// TIA Portal V20 export
// export: Created 2025-12-01T14:56:17.5233973Z, ExportSetting None, DisplayName Totally Integrated Automation Portal, DisplayVersion V20 Update 3, DisplayName TIA Portal Openness, DisplayVersion V20 Update 3, DisplayName TIA Portal Version Control Interface, DisplayVersion V20 Update 3, DisplayName STEP 7 Professional, DisplayVersion V20 Update 3, DisplayName STEP 7 Safety, DisplayVersion V20 Update 2, DisplayName WinCC Basic/Comfort/Advanced, DisplayVersion V20 Update 3, DisplayName WinCC Professional, DisplayVersion V20 Update 3, DisplayName WinCC Unified, DisplayVersion V20 Update 3
TYPE "Interlock_QubiqaUlma"
   STRUCT
      TL_Online { ExternalVisible := 'False'} : Bool;
      TL_Alive { ExternalVisible := 'False'} : Bool;
      TL1_Run { ExternalVisible := 'False'} : Bool;
      TL2_Run { ExternalVisible := 'False'} : Bool;
      TL1_StartButton { ExternalVisible := 'False'} : Bool;
      TL1_ResetButton { ExternalVisible := 'False'} : Bool;
      TL2_StartButton { ExternalVisible := 'False'} : Bool;
      TL2_ResetButton { ExternalVisible := 'False'} : Bool;
      Reserve_1_0 { ExternalVisible := 'False'} : Bool;
      Reserve_1_1 { ExternalVisible := 'False'} : Bool;
      Reserve_1_2 { ExternalVisible := 'False'} : Bool;
      Reserve_1_3 { ExternalVisible := 'False'} : Bool;
      Reserve_1_4 { ExternalVisible := 'False'} : Bool;
      Reserve_1_5 { ExternalVisible := 'False'} : Bool;
      Reserve_1_6 { ExternalVisible := 'False'} : Bool;
      Reserve_1_7 { ExternalVisible := 'False'} : Bool;
      LineRunning_L1 { ExternalVisible := 'False'} : Bool;
      TrayInTransfer_L1 { ExternalVisible := 'False'} : Bool;
      SorterInductionSpeed_L1 { ExternalVisible := 'False'} : Bool;
      SizeControl_L1 { ExternalVisible := 'False'} : Bool;
      Reserve_2_4 { ExternalVisible := 'False'} : Bool;
      Reserve_2_5 { ExternalVisible := 'False'} : Bool;
      Reserve_2_6 { ExternalVisible := 'False'} : Bool;
      OrderFinished_L1 { ExternalVisible := 'False'} : Bool;
      PermissionToSend_L1 { ExternalVisible := 'False'} : Bool;
      TranserFinished_L1 { ExternalVisible := 'False'} : Bool;
      OrderFinished_Ok_L1 { ExternalVisible := 'False'} : Bool;
      reserva_3_3 { ExternalVisible := 'False'} : Bool;
      reserva_3_4 { ExternalVisible := 'False'} : Bool;
      reserva_3_5 { ExternalVisible := 'False'} : Bool;
      reserva_3_6 { ExternalVisible := 'False'} : Bool;
      reserva_3_7 { ExternalVisible := 'False'} : Bool;
      StartStack_Small_L1 { ExternalVisible := 'False'} : Bool;
      StackReceived_Small_L1 { ExternalVisible := 'False'} : Bool;
      reserva_4_2 { ExternalVisible := 'False'} : Bool;
      reserva_4_3 { ExternalVisible := 'False'} : Bool;
      reserva_4_4 { ExternalVisible := 'False'} : Bool;
      reserva_4_5 { ExternalVisible := 'False'} : Bool;
      reserva_4_6 { ExternalVisible := 'False'} : Bool;
      reserva_4_7 { ExternalVisible := 'False'} : Bool;
      NoStackInBuffer_Small_L1 { ExternalVisible := 'False'} : Byte;
      StartStack_Large_L1 { ExternalVisible := 'False'} : Bool;
      StackReceived_Large_L1 { ExternalVisible := 'False'} : Bool;
      reserva_6_2 { ExternalVisible := 'False'} : Bool;
      reserva_6_3 { ExternalVisible := 'False'} : Bool;
      reserva_6_4 { ExternalVisible := 'False'} : Bool;
      reserva_6_5 { ExternalVisible := 'False'} : Bool;
      reserva_6_6 { ExternalVisible := 'False'} : Bool;
      reserva_6_7 { ExternalVisible := 'False'} : Bool;
      NoStackInBuffer_Large_L1 { ExternalVisible := 'False'} : Byte;
      reserva_8_0 { ExternalVisible := 'False'} : Bool;
      reserva_8_1 { ExternalVisible := 'False'} : Bool;
      reserva_8_2 { ExternalVisible := 'False'} : Bool;
      reserva_8_3 { ExternalVisible := 'False'} : Bool;
      reserva_8_4 { ExternalVisible := 'False'} : Bool;
      reserva_8_5 { ExternalVisible := 'False'} : Bool;
      reserva_8_6 { ExternalVisible := 'False'} : Bool;
      reserva_8_7 { ExternalVisible := 'False'} : Bool;
      reserva_9_0 { ExternalVisible := 'False'} : Bool;
      reserva_9_1 { ExternalVisible := 'False'} : Bool;
      reserva_9_2 { ExternalVisible := 'False'} : Bool;
      reserva_9_3 { ExternalVisible := 'False'} : Bool;
      reserva_9_4 { ExternalVisible := 'False'} : Bool;
      reserva_9_5 { ExternalVisible := 'False'} : Bool;
      reserva_9_6 { ExternalVisible := 'False'} : Bool;
      reserva_9_7 { ExternalVisible := 'False'} : Bool;
      LineRunning_L2 { ExternalVisible := 'False'} : Bool;
      TrayInTransfer_L2 { ExternalVisible := 'False'} : Bool;
      SorterInductionSpeed_L2 { ExternalVisible := 'False'} : Bool;
      SizeControl_L2 { ExternalVisible := 'False'} : Bool;
      reserva_10_4 { ExternalVisible := 'False'} : Bool;
      reserva_10_5 { ExternalVisible := 'False'} : Bool;
      reserva_10_6 { ExternalVisible := 'False'} : Bool;
      OrderFinished_L2 { ExternalVisible := 'False'} : Bool;
      PermissionToSend_L2 { ExternalVisible := 'False'} : Bool;
      TranserFinished_L2 { ExternalVisible := 'False'} : Bool;
      OrderFinished_Ok_L2 { ExternalVisible := 'False'} : Bool;
      reserva_11_3 { ExternalVisible := 'False'} : Bool;
      reserva_11_4 { ExternalVisible := 'False'} : Bool;
      reserva_11_5 { ExternalVisible := 'False'} : Bool;
      reserva_11_6 { ExternalVisible := 'False'} : Bool;
      reserva_11_7 { ExternalVisible := 'False'} : Bool;
      StartStack_Small_L2 { ExternalVisible := 'False'} : Bool;
      StackReceived_Small_L2 { ExternalVisible := 'False'} : Bool;
      reserva_12_2 { ExternalVisible := 'False'} : Bool;
      reserva_12_3 { ExternalVisible := 'False'} : Bool;
      reserva_12_4 { ExternalVisible := 'False'} : Bool;
      reserva_12_5 { ExternalVisible := 'False'} : Bool;
      reserva_12_6 { ExternalVisible := 'False'} : Bool;
      reserva_12_7 { ExternalVisible := 'False'} : Bool;
      NoStackInBuffer_Small_L2 { ExternalVisible := 'False'} : Byte;
      StartStack_Large_L2 { ExternalVisible := 'False'} : Bool;
      StackReceived_Large_L2 { ExternalVisible := 'False'} : Bool;
      reserva_14_2 { ExternalVisible := 'False'} : Bool;
      reserva_14_3 { ExternalVisible := 'False'} : Bool;
      reserva_14_4 { ExternalVisible := 'False'} : Bool;
      reserva_14_5 { ExternalVisible := 'False'} : Bool;
      reserva_14_6 { ExternalVisible := 'False'} : Bool;
      reserva_14_7 { ExternalVisible := 'False'} : Bool;
      NoStackInBuffer_Large_L2 { ExternalVisible := 'False'} : Byte;
      reserva_16_0 { ExternalVisible := 'False'} : Bool;
      reserva_16_1 { ExternalVisible := 'False'} : Bool;
      reserva_16_2 { ExternalVisible := 'False'} : Bool;
      reserva_16_3 { ExternalVisible := 'False'} : Bool;
      reserva_16_4 { ExternalVisible := 'False'} : Bool;
      reserva_16_5 { ExternalVisible := 'False'} : Bool;
      reserva_16_6 { ExternalVisible := 'False'} : Bool;
      reserva_16_7 { ExternalVisible := 'False'} : Bool;
      reserva_17_0 { ExternalVisible := 'False'} : Bool;
      reserva_17_1 { ExternalVisible := 'False'} : Bool;
      reserva_17_2 { ExternalVisible := 'False'} : Bool;
      reserva_17_3 { ExternalVisible := 'False'} : Bool;
      reserva_17_4 { ExternalVisible := 'False'} : Bool;
      reserva_17_5 { ExternalVisible := 'False'} : Bool;
      reserva_17_6 { ExternalVisible := 'False'} : Bool;
      reserva_17_7 { ExternalVisible := 'False'} : Bool;
      reserva_18_0 { ExternalVisible := 'False'} : Bool;
      reserva_18_1 { ExternalVisible := 'False'} : Bool;
      reserva_18_2 { ExternalVisible := 'False'} : Bool;
      reserva_18_3 { ExternalVisible := 'False'} : Bool;
      reserva_18_4 { ExternalVisible := 'False'} : Bool;
      reserva_18_5 { ExternalVisible := 'False'} : Bool;
      reserva_18_6 { ExternalVisible := 'False'} : Bool;
      reserva_18_7 { ExternalVisible := 'False'} : Bool;
      reserva_19_0 { ExternalVisible := 'False'} : Bool;
      reserva_19_1 { ExternalVisible := 'False'} : Bool;
      reserva_19_2 { ExternalVisible := 'False'} : Bool;
      reserva_19_3 { ExternalVisible := 'False'} : Bool;
      reserva_19_4 { ExternalVisible := 'False'} : Bool;
      reserva_19_5 { ExternalVisible := 'False'} : Bool;
      reserva_19_6 { ExternalVisible := 'False'} : Bool;
      reserva_19_7 { ExternalVisible := 'False'} : Bool;
      reserva_20_0 { ExternalVisible := 'False'} : Bool;
      reserva_20_1 { ExternalVisible := 'False'} : Bool;
      reserva_20_2 { ExternalVisible := 'False'} : Bool;
      reserva_20_3 { ExternalVisible := 'False'} : Bool;
      reserva_20_4 { ExternalVisible := 'False'} : Bool;
      reserva_20_5 { ExternalVisible := 'False'} : Bool;
      reserva_20_6 { ExternalVisible := 'False'} : Bool;
      reserva_20_7 { ExternalVisible := 'False'} : Bool;
      reserva_21_0 { ExternalVisible := 'False'} : Bool;
      reserva_21_1 { ExternalVisible := 'False'} : Bool;
      reserva_21_2 { ExternalVisible := 'False'} : Bool;
      reserva_21_3 { ExternalVisible := 'False'} : Bool;
      reserva_21_4 { ExternalVisible := 'False'} : Bool;
      reserva_21_5 { ExternalVisible := 'False'} : Bool;
      reserva_21_6 { ExternalVisible := 'False'} : Bool;
      reserva_21_7 { ExternalVisible := 'False'} : Bool;
      reserva_22_0 { ExternalVisible := 'False'} : Bool;
      reserva_22_1 { ExternalVisible := 'False'} : Bool;
      reserva_22_2 { ExternalVisible := 'False'} : Bool;
      reserva_22_3 { ExternalVisible := 'False'} : Bool;
      reserva_22_4 { ExternalVisible := 'False'} : Bool;
      reserva_22_5 { ExternalVisible := 'False'} : Bool;
      reserva_22_6 { ExternalVisible := 'False'} : Bool;
      reserva_22_7 { ExternalVisible := 'False'} : Bool;
      reserva_23_0 { ExternalVisible := 'False'} : Bool;
      reserva_23_1 { ExternalVisible := 'False'} : Bool;
      reserva_23_2 { ExternalVisible := 'False'} : Bool;
      reserva_23_3 { ExternalVisible := 'False'} : Bool;
      reserva_23_4 { ExternalVisible := 'False'} : Bool;
      reserva_23_5 { ExternalVisible := 'False'} : Bool;
      reserva_23_6 { ExternalVisible := 'False'} : Bool;
      reserva_23_7 { ExternalVisible := 'False'} : Bool;
      reserva_24_0 { ExternalVisible := 'False'} : Bool;
      reserva_24_1 { ExternalVisible := 'False'} : Bool;
      reserva_24_2 { ExternalVisible := 'False'} : Bool;
      reserva_24_3 { ExternalVisible := 'False'} : Bool;
      reserva_24_4 { ExternalVisible := 'False'} : Bool;
      reserva_24_5 { ExternalVisible := 'False'} : Bool;
      reserva_24_6 { ExternalVisible := 'False'} : Bool;
      reserva_24_7 { ExternalVisible := 'False'} : Bool;
      reserva_25_0 { ExternalVisible := 'False'} : Bool;
      reserva_25_1 { ExternalVisible := 'False'} : Bool;
      reserva_25_2 { ExternalVisible := 'False'} : Bool;
      reserva_25_3 { ExternalVisible := 'False'} : Bool;
      reserva_25_4 { ExternalVisible := 'False'} : Bool;
      reserva_25_5 { ExternalVisible := 'False'} : Bool;
      reserva_25_6 { ExternalVisible := 'False'} : Bool;
      reserva_25_7 { ExternalVisible := 'False'} : Bool;
      reserva_26_0 { ExternalVisible := 'False'} : Bool;
      reserva_26_1 { ExternalVisible := 'False'} : Bool;
      reserva_26_2 { ExternalVisible := 'False'} : Bool;
      reserva_26_3 { ExternalVisible := 'False'} : Bool;
      reserva_26_4 { ExternalVisible := 'False'} : Bool;
      reserva_26_5 { ExternalVisible := 'False'} : Bool;
      reserva_26_6 { ExternalVisible := 'False'} : Bool;
      reserva_26_7 { ExternalVisible := 'False'} : Bool;
      reserva_27_0 { ExternalVisible := 'False'} : Bool;
      reserva_27_1 { ExternalVisible := 'False'} : Bool;
      reserva_27_2 { ExternalVisible := 'False'} : Bool;
      reserva_27_3 { ExternalVisible := 'False'} : Bool;
      reserva_27_4 { ExternalVisible := 'False'} : Bool;
      reserva_27_5 { ExternalVisible := 'False'} : Bool;
      reserva_27_6 { ExternalVisible := 'False'} : Bool;
      reserva_27_7 { ExternalVisible := 'False'} : Bool;
      reserva_28_0 { ExternalVisible := 'False'} : Bool;
      reserva_28_1 { ExternalVisible := 'False'} : Bool;
      reserva_28_2 { ExternalVisible := 'False'} : Bool;
      reserva_28_3 { ExternalVisible := 'False'} : Bool;
      reserva_28_4 { ExternalVisible := 'False'} : Bool;
      reserva_28_5 { ExternalVisible := 'False'} : Bool;
      reserva_28_6 { ExternalVisible := 'False'} : Bool;
      reserva_28_7 { ExternalVisible := 'False'} : Bool;
      reserva_29_0 { ExternalVisible := 'False'} : Bool;
      reserva_29_1 { ExternalVisible := 'False'} : Bool;
      reserva_29_2 { ExternalVisible := 'False'} : Bool;
      reserva_29_3 { ExternalVisible := 'False'} : Bool;
      reserva_29_4 { ExternalVisible := 'False'} : Bool;
      reserva_29_5 { ExternalVisible := 'False'} : Bool;
      reserva_29_6 { ExternalVisible := 'False'} : Bool;
      reserva_29_7 { ExternalVisible := 'False'} : Bool;
      Reserve_30_0 { ExternalVisible := 'False'} : Bool;
      Reserve_30_1 { ExternalVisible := 'False'} : Bool;
      Reserve_30_2 { ExternalVisible := 'False'} : Bool;
      Reserve_30_3 { ExternalVisible := 'False'} : Bool;
      Reserve_30_4 { ExternalVisible := 'False'} : Bool;
      Reserve_30_5 { ExternalVisible := 'False'} : Bool;
      Reserve_30_6 { ExternalVisible := 'False'} : Bool;
      Reserve_30_7 { ExternalVisible := 'False'} : Bool;
      Reserve_31_0 { ExternalVisible := 'False'} : Bool;
      Reserve_31_1 { ExternalVisible := 'False'} : Bool;
      Reserve_31_2 { ExternalVisible := 'False'} : Bool;
      Reserve_31_3 { ExternalVisible := 'False'} : Bool;
      Reserve_31_4 { ExternalVisible := 'False'} : Bool;
      Reserve_31_5 { ExternalVisible := 'False'} : Bool;
      Reserve_31_6 { ExternalVisible := 'False'} : Bool;
      Reserve_31_7 { ExternalVisible := 'False'} : Bool;
      Reserve_32_0 { ExternalVisible := 'False'} : Bool;
      Reserve_32_1 { ExternalVisible := 'False'} : Bool;
      Reserve_32_2 { ExternalVisible := 'False'} : Bool;
      Reserve_32_3 { ExternalVisible := 'False'} : Bool;
      Reserve_32_4 { ExternalVisible := 'False'} : Bool;
      Reserve_32_5 { ExternalVisible := 'False'} : Bool;
      Reserve_32_6 { ExternalVisible := 'False'} : Bool;
      Reserve_32_7 { ExternalVisible := 'False'} : Bool;
      reserva_33_0 { ExternalVisible := 'False'} : Bool;
      reserva_33_1 { ExternalVisible := 'False'} : Bool;
      reserva_33_2 { ExternalVisible := 'False'} : Bool;
      reserva_33_3 { ExternalVisible := 'False'} : Bool;
      reserva_33_4 { ExternalVisible := 'False'} : Bool;
      reserva_33_5 { ExternalVisible := 'False'} : Bool;
      reserva_33_6 { ExternalVisible := 'False'} : Bool;
      reserva_33_7 { ExternalVisible := 'False'} : Bool;
      reserva_34_0 { ExternalVisible := 'False'} : Bool;
      reserva_34_1 { ExternalVisible := 'False'} : Bool;
      reserva_34_2 { ExternalVisible := 'False'} : Bool;
      reserva_34_3 { ExternalVisible := 'False'} : Bool;
      reserva_34_4 { ExternalVisible := 'False'} : Bool;
      reserva_34_5 { ExternalVisible := 'False'} : Bool;
      reserva_34_6 { ExternalVisible := 'False'} : Bool;
      reserva_34_7 { ExternalVisible := 'False'} : Bool;
      reserva_35_0 { ExternalVisible := 'False'} : Bool;
      reserva_35_1 { ExternalVisible := 'False'} : Bool;
      reserva_35_2 { ExternalVisible := 'False'} : Bool;
      reserva_35_3 { ExternalVisible := 'False'} : Bool;
      reserva_35_4 { ExternalVisible := 'False'} : Bool;
      reserva_35_5 { ExternalVisible := 'False'} : Bool;
      reserva_35_6 { ExternalVisible := 'False'} : Bool;
      reserva_35_7 { ExternalVisible := 'False'} : Bool;
      reserva_36_0 { ExternalVisible := 'False'} : Bool;
      reserva_36_1 { ExternalVisible := 'False'} : Bool;
      reserva_36_2 { ExternalVisible := 'False'} : Bool;
      reserva_36_3 { ExternalVisible := 'False'} : Bool;
      reserva_36_4 { ExternalVisible := 'False'} : Bool;
      reserva_36_5 { ExternalVisible := 'False'} : Bool;
      reserva_36_6 { ExternalVisible := 'False'} : Bool;
      reserva_36_7 { ExternalVisible := 'False'} : Bool;
      reserva_37_0 { ExternalVisible := 'False'} : Bool;
      reserva_37_1 { ExternalVisible := 'False'} : Bool;
      reserva_37_2 { ExternalVisible := 'False'} : Bool;
      reserva_37_3 { ExternalVisible := 'False'} : Bool;
      reserva_37_4 { ExternalVisible := 'False'} : Bool;
      reserva_37_5 { ExternalVisible := 'False'} : Bool;
      reserva_37_6 { ExternalVisible := 'False'} : Bool;
      reserva_37_7 { ExternalVisible := 'False'} : Bool;
      reserva_38_0 { ExternalVisible := 'False'} : Bool;
      reserva_38_1 { ExternalVisible := 'False'} : Bool;
      reserva_38_2 { ExternalVisible := 'False'} : Bool;
      reserva_38_3 { ExternalVisible := 'False'} : Bool;
      reserva_38_4 { ExternalVisible := 'False'} : Bool;
      reserva_38_5 { ExternalVisible := 'False'} : Bool;
      reserva_38_6 { ExternalVisible := 'False'} : Bool;
      reserva_38_7 { ExternalVisible := 'False'} : Bool;
      reserva_39_0 { ExternalVisible := 'False'} : Bool;
      reserva_39_1 { ExternalVisible := 'False'} : Bool;
      reserva_39_2 { ExternalVisible := 'False'} : Bool;
      reserva_39_3 { ExternalVisible := 'False'} : Bool;
      reserva_39_4 { ExternalVisible := 'False'} : Bool;
      reserva_39_5 { ExternalVisible := 'False'} : Bool;
      reserva_39_6 { ExternalVisible := 'False'} : Bool;
      reserva_39_7 { ExternalVisible := 'False'} : Bool;
      reserva_40_0 { ExternalVisible := 'False'} : Bool;
      reserva_40_1 { ExternalVisible := 'False'} : Bool;
      reserva_40_2 { ExternalVisible := 'False'} : Bool;
      reserva_40_3 { ExternalVisible := 'False'} : Bool;
      reserva_40_4 { ExternalVisible := 'False'} : Bool;
      reserva_40_5 { ExternalVisible := 'False'} : Bool;
      reserva_40_6 { ExternalVisible := 'False'} : Bool;
      reserva_40_7 { ExternalVisible := 'False'} : Bool;
      reserva_41_0 { ExternalVisible := 'False'} : Bool;
      reserva_41_1 { ExternalVisible := 'False'} : Bool;
      reserva_41_2 { ExternalVisible := 'False'} : Bool;
      reserva_41_3 { ExternalVisible := 'False'} : Bool;
      reserva_41_4 { ExternalVisible := 'False'} : Bool;
      reserva_41_5 { ExternalVisible := 'False'} : Bool;
      reserva_41_6 { ExternalVisible := 'False'} : Bool;
      reserva_41_7 { ExternalVisible := 'False'} : Bool;
      reserva_42_0 { ExternalVisible := 'False'} : Bool;
      reserva_42_1 { ExternalVisible := 'False'} : Bool;
      reserva_42_2 { ExternalVisible := 'False'} : Bool;
      reserva_42_3 { ExternalVisible := 'False'} : Bool;
      reserva_42_4 { ExternalVisible := 'False'} : Bool;
      reserva_42_5 { ExternalVisible := 'False'} : Bool;
      reserva_42_6 { ExternalVisible := 'False'} : Bool;
      reserva_42_7 { ExternalVisible := 'False'} : Bool;
      reserva_43_0 { ExternalVisible := 'False'} : Bool;
      reserva_43_1 { ExternalVisible := 'False'} : Bool;
      reserva_43_2 { ExternalVisible := 'False'} : Bool;
      reserva_43_3 { ExternalVisible := 'False'} : Bool;
      reserva_43_4 { ExternalVisible := 'False'} : Bool;
      reserva_43_5 { ExternalVisible := 'False'} : Bool;
      reserva_43_6 { ExternalVisible := 'False'} : Bool;
      reserva_43_7 { ExternalVisible := 'False'} : Bool;
      reserva_44_0 { ExternalVisible := 'False'} : Bool;
      reserva_44_1 { ExternalVisible := 'False'} : Bool;
      reserva_44_2 { ExternalVisible := 'False'} : Bool;
      reserva_44_3 { ExternalVisible := 'False'} : Bool;
      reserva_44_4 { ExternalVisible := 'False'} : Bool;
      reserva_44_5 { ExternalVisible := 'False'} : Bool;
      reserva_44_6 { ExternalVisible := 'False'} : Bool;
      reserva_44_7 { ExternalVisible := 'False'} : Bool;
      reserva_45_0 { ExternalVisible := 'False'} : Bool;
      reserva_45_1 { ExternalVisible := 'False'} : Bool;
      reserva_45_2 { ExternalVisible := 'False'} : Bool;
      reserva_45_3 { ExternalVisible := 'False'} : Bool;
      reserva_45_4 { ExternalVisible := 'False'} : Bool;
      reserva_45_5 { ExternalVisible := 'False'} : Bool;
      reserva_45_6 { ExternalVisible := 'False'} : Bool;
      reserva_45_7 { ExternalVisible := 'False'} : Bool;
      reserva_46_0 { ExternalVisible := 'False'} : Bool;
      reserva_46_1 { ExternalVisible := 'False'} : Bool;
      reserva_46_2 { ExternalVisible := 'False'} : Bool;
      reserva_46_3 { ExternalVisible := 'False'} : Bool;
      reserva_46_4 { ExternalVisible := 'False'} : Bool;
      reserva_46_5 { ExternalVisible := 'False'} : Bool;
      reserva_46_6 { ExternalVisible := 'False'} : Bool;
      reserva_46_7 { ExternalVisible := 'False'} : Bool;
      reserva_47_0 { ExternalVisible := 'False'} : Bool;
      reserva_47_1 { ExternalVisible := 'False'} : Bool;
      reserva_47_2 { ExternalVisible := 'False'} : Bool;
      reserva_47_3 { ExternalVisible := 'False'} : Bool;
      reserva_47_4 { ExternalVisible := 'False'} : Bool;
      reserva_47_5 { ExternalVisible := 'False'} : Bool;
      reserva_47_6 { ExternalVisible := 'False'} : Bool;
      reserva_47_7 { ExternalVisible := 'False'} : Bool;
      reserva_48_0 { ExternalVisible := 'False'} : Bool;
      reserva_48_1 { ExternalVisible := 'False'} : Bool;
      reserva_48_2 { ExternalVisible := 'False'} : Bool;
      reserva_48_3 { ExternalVisible := 'False'} : Bool;
      reserva_48_4 { ExternalVisible := 'False'} : Bool;
      reserva_48_5 { ExternalVisible := 'False'} : Bool;
      reserva_48_6 { ExternalVisible := 'False'} : Bool;
      reserva_48_7 { ExternalVisible := 'False'} : Bool;
      reserva_49_0 { ExternalVisible := 'False'} : Bool;
      reserva_49_1 { ExternalVisible := 'False'} : Bool;
      reserva_49_2 { ExternalVisible := 'False'} : Bool;
      reserva_49_3 { ExternalVisible := 'False'} : Bool;
      reserva_49_4 { ExternalVisible := 'False'} : Bool;
      reserva_49_5 { ExternalVisible := 'False'} : Bool;
      reserva_49_6 { ExternalVisible := 'False'} : Bool;
      reserva_49_7 { ExternalVisible := 'False'} : Bool;
      reserva_50_0 { ExternalVisible := 'False'} : Bool;
      reserva_50_1 { ExternalVisible := 'False'} : Bool;
      reserva_50_2 { ExternalVisible := 'False'} : Bool;
      reserva_50_3 { ExternalVisible := 'False'} : Bool;
      reserva_50_4 { ExternalVisible := 'False'} : Bool;
      reserva_50_5 { ExternalVisible := 'False'} : Bool;
      reserva_50_6 { ExternalVisible := 'False'} : Bool;
      reserva_50_7 { ExternalVisible := 'False'} : Bool;
      reserva_51_0 { ExternalVisible := 'False'} : Bool;
      reserva_51_1 { ExternalVisible := 'False'} : Bool;
      reserva_51_2 { ExternalVisible := 'False'} : Bool;
      reserva_51_3 { ExternalVisible := 'False'} : Bool;
      reserva_51_4 { ExternalVisible := 'False'} : Bool;
      reserva_51_5 { ExternalVisible := 'False'} : Bool;
      reserva_51_6 { ExternalVisible := 'False'} : Bool;
      reserva_51_7 { ExternalVisible := 'False'} : Bool;
      reserva_52_0 { ExternalVisible := 'False'} : Bool;
      reserva_52_1 { ExternalVisible := 'False'} : Bool;
      reserva_52_2 { ExternalVisible := 'False'} : Bool;
      reserva_52_3 { ExternalVisible := 'False'} : Bool;
      reserva_52_4 { ExternalVisible := 'False'} : Bool;
      reserva_52_5 { ExternalVisible := 'False'} : Bool;
      reserva_52_6 { ExternalVisible := 'False'} : Bool;
      reserva_52_7 { ExternalVisible := 'False'} : Bool;
      reserva_53_0 { ExternalVisible := 'False'} : Bool;
      reserva_53_1 { ExternalVisible := 'False'} : Bool;
      reserva_53_2 { ExternalVisible := 'False'} : Bool;
      reserva_53_3 { ExternalVisible := 'False'} : Bool;
      reserva_53_4 { ExternalVisible := 'False'} : Bool;
      reserva_53_5 { ExternalVisible := 'False'} : Bool;
      reserva_53_6 { ExternalVisible := 'False'} : Bool;
      reserva_53_7 { ExternalVisible := 'False'} : Bool;
      reserva_54_0 { ExternalVisible := 'False'} : Bool;
      reserva_54_1 { ExternalVisible := 'False'} : Bool;
      reserva_54_2 { ExternalVisible := 'False'} : Bool;
      reserva_54_3 { ExternalVisible := 'False'} : Bool;
      reserva_54_4 { ExternalVisible := 'False'} : Bool;
      reserva_54_5 { ExternalVisible := 'False'} : Bool;
      reserva_54_6 { ExternalVisible := 'False'} : Bool;
      reserva_54_7 { ExternalVisible := 'False'} : Bool;
      reserva_55_0 { ExternalVisible := 'False'} : Bool;
      reserva_55_1 { ExternalVisible := 'False'} : Bool;
      reserva_55_2 { ExternalVisible := 'False'} : Bool;
      reserva_55_3 { ExternalVisible := 'False'} : Bool;
      reserva_55_4 { ExternalVisible := 'False'} : Bool;
      reserva_55_5 { ExternalVisible := 'False'} : Bool;
      reserva_55_6 { ExternalVisible := 'False'} : Bool;
      reserva_55_7 { ExternalVisible := 'False'} : Bool;
      reserva_56_0 { ExternalVisible := 'False'} : Bool;
      reserva_56_1 { ExternalVisible := 'False'} : Bool;
      reserva_56_2 { ExternalVisible := 'False'} : Bool;
      reserva_56_3 { ExternalVisible := 'False'} : Bool;
      reserva_56_4 { ExternalVisible := 'False'} : Bool;
      reserva_56_5 { ExternalVisible := 'False'} : Bool;
      reserva_56_6 { ExternalVisible := 'False'} : Bool;
      reserva_56_7 { ExternalVisible := 'False'} : Bool;
      reserva_57_0 { ExternalVisible := 'False'} : Bool;
      reserva_57_1 { ExternalVisible := 'False'} : Bool;
      reserva_57_2 { ExternalVisible := 'False'} : Bool;
      reserva_57_3 { ExternalVisible := 'False'} : Bool;
      reserva_57_4 { ExternalVisible := 'False'} : Bool;
      reserva_57_5 { ExternalVisible := 'False'} : Bool;
      reserva_57_6 { ExternalVisible := 'False'} : Bool;
      reserva_57_7 { ExternalVisible := 'False'} : Bool;
      reserva_58_0 { ExternalVisible := 'False'} : Bool;
      reserva_58_1 { ExternalVisible := 'False'} : Bool;
      reserva_58_2 { ExternalVisible := 'False'} : Bool;
      reserva_58_3 { ExternalVisible := 'False'} : Bool;
      reserva_58_4 { ExternalVisible := 'False'} : Bool;
      reserva_58_5 { ExternalVisible := 'False'} : Bool;
      reserva_58_6 { ExternalVisible := 'False'} : Bool;
      reserva_58_7 { ExternalVisible := 'False'} : Bool;
      reserva_59_0 { ExternalVisible := 'False'} : Bool;
      reserva_59_1 { ExternalVisible := 'False'} : Bool;
      reserva_59_2 { ExternalVisible := 'False'} : Bool;
      reserva_59_3 { ExternalVisible := 'False'} : Bool;
      reserva_59_4 { ExternalVisible := 'False'} : Bool;
      reserva_59_5 { ExternalVisible := 'False'} : Bool;
      reserva_59_6 { ExternalVisible := 'False'} : Bool;
      reserva_59_7 { ExternalVisible := 'False'} : Bool;
      Reserve_60_0 { ExternalVisible := 'False'} : Bool;
      Reserve_60_1 { ExternalVisible := 'False'} : Bool;
      Reserve_60_2 { ExternalVisible := 'False'} : Bool;
      Reserve_60_3 { ExternalVisible := 'False'} : Bool;
      Reserve_60_4 { ExternalVisible := 'False'} : Bool;
      Reserve_60_5 { ExternalVisible := 'False'} : Bool;
      Reserve_60_6 { ExternalVisible := 'False'} : Bool;
      Reserve_60_7 { ExternalVisible := 'False'} : Bool;
      reserva_61_0 { ExternalVisible := 'False'} : Bool;
      reserva_61_1 { ExternalVisible := 'False'} : Bool;
      reserva_61_2 { ExternalVisible := 'False'} : Bool;
      reserva_61_3 { ExternalVisible := 'False'} : Bool;
      reserva_61_4 { ExternalVisible := 'False'} : Bool;
      reserva_61_5 { ExternalVisible := 'False'} : Bool;
      reserva_61_6 { ExternalVisible := 'False'} : Bool;
      reserva_61_7 { ExternalVisible := 'False'} : Bool;
      Reserve_62_0 { ExternalVisible := 'False'} : Bool;
      Reserve_62_1 { ExternalVisible := 'False'} : Bool;
      Reserve_62_2 { ExternalVisible := 'False'} : Bool;
      Reserve_62_3 { ExternalVisible := 'False'} : Bool;
      Reserve_62_4 { ExternalVisible := 'False'} : Bool;
      Reserve_62_5 { ExternalVisible := 'False'} : Bool;
      Reserve_62_6 { ExternalVisible := 'False'} : Bool;
      Reserve_62_7 { ExternalVisible := 'False'} : Bool;
      Reserve_63_0 { ExternalVisible := 'False'} : Bool;
      Reserve_63_1 { ExternalVisible := 'False'} : Bool;
      Reserve_63_2 { ExternalVisible := 'False'} : Bool;
      Reserve_63_3 { ExternalVisible := 'False'} : Bool;
      Reserve_63_4 { ExternalVisible := 'False'} : Bool;
      Reserve_63_5 { ExternalVisible := 'False'} : Bool;
      Reserve_63_6 { ExternalVisible := 'False'} : Bool;
      Reserve_63_7 { ExternalVisible := 'False'} : Bool;
      Reserve_64_0 { ExternalVisible := 'False'} : Bool;
      Reserve_64_1 { ExternalVisible := 'False'} : Bool;
      Reserve_64_2 { ExternalVisible := 'False'} : Bool;
      Reserve_64_3 { ExternalVisible := 'False'} : Bool;
      Reserve_64_4 { ExternalVisible := 'False'} : Bool;
      Reserve_64_5 { ExternalVisible := 'False'} : Bool;
      Reserve_64_6 { ExternalVisible := 'False'} : Bool;
      Reserve_64_7 { ExternalVisible := 'False'} : Bool;
      Reserve_65_0 { ExternalVisible := 'False'} : Bool;
      Reserve_65_1 { ExternalVisible := 'False'} : Bool;
      Reserve_65_2 { ExternalVisible := 'False'} : Bool;
      Reserve_65_3 { ExternalVisible := 'False'} : Bool;
      Reserve_65_4 { ExternalVisible := 'False'} : Bool;
      Reserve_65_5 { ExternalVisible := 'False'} : Bool;
      Reserve_65_6 { ExternalVisible := 'False'} : Bool;
      Reserve_65_7 { ExternalVisible := 'False'} : Bool;
   END_STRUCT;
END_TYPE
